// Mitsubishi GX Works2 project: ratanak_farm10   PLC: FX3U/FX3UC

PROGRAM MAIN
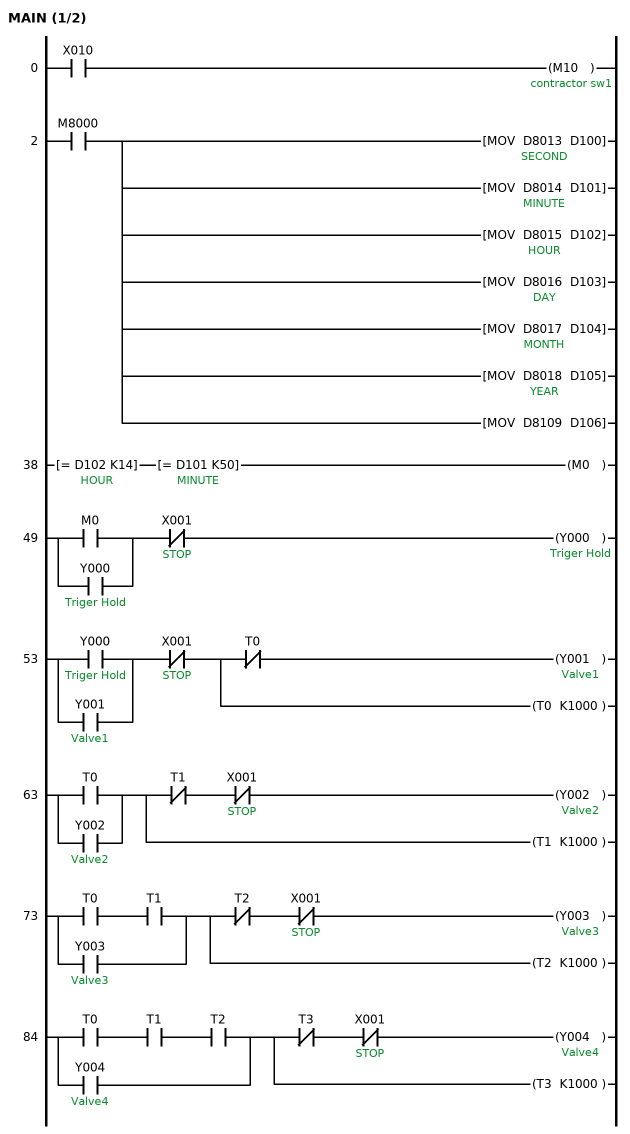
0     LD      X010
      OUT     M10  ; contractor sw1
2     LD      M8000
      MOV     D8013 D100  ; SECOND
      MOV     D8014 D101  ; MINUTE
      MOV     D8015 D102  ; HOUR
      MOV     D8016 D103  ; DAY
      MOV     D8017 D104  ; MONTH
      MOV     D8018 D105  ; YEAR
      MOV     D8109 D106
38    LD=     D102 K14  ; HOUR
      AND=    D101 K50  ; MINUTE
      OUT     M0
49    LD      M0
      OR      Y000  ; Triger Hold
      ANI     X001  ; STOP
      OUT     Y000  ; Triger Hold
53    LD      Y000  ; Triger Hold
      OR      Y001  ; Valve1
      ANI     X001  ; STOP
      MPS
      ANI     T0
      OUT     Y001  ; Valve1
      MPP
      OUT     T0 K1000
63    LD      T0
      OR      Y002  ; Valve2
      MPS
      ANI     T1
      ANI     X001  ; STOP
      OUT     Y002  ; Valve2
      MPP
      OUT     T1 K1000
73    LD      T0
      AND     T1
      OR      Y003  ; Valve3
      MPS
      ANI     T2
      ANI     X001  ; STOP
      OUT     Y003  ; Valve3
      MPP
      OUT     T2 K1000
84    LD      T0
      AND     T1
      AND     T2
      OR      Y004  ; Valve4
      MPS
      ANI     T3
      ANI     X001  ; STOP
      OUT     Y004  ; Valve4
      MPP
      OUT     T3 K1000
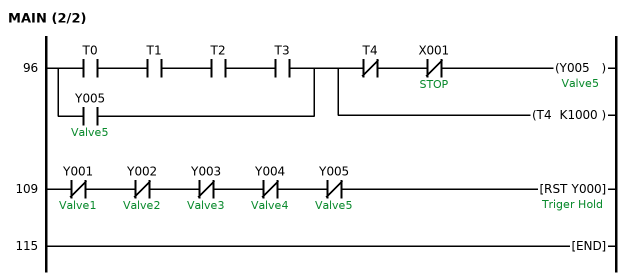
96    LD      T0
      AND     T1
      AND     T2
      AND     T3
      OR      Y005  ; Valve5
      MPS
      ANI     T4
      ANI     X001  ; STOP
      OUT     Y005  ; Valve5
      MPP
      OUT     T4 K1000
109   LDI     Y001  ; Valve1
      ANI     Y002  ; Valve2
      ANI     Y003  ; Valve3
      ANI     Y004  ; Valve4
      ANI     Y005  ; Valve5
      RST     Y000  ; Triger Hold
115   END
END_PROGRAM

// device comments not shown above
X000  ; START
M11  ; contractor sw2
